      L     #WT_Nr;  //Warenträger-DB öffnen
      L     100;
      +I;
      T     #WT_DB;
      OPN   DB [#WT_DB];
      L     #WT_Nr_lang;
      T     "DB_BE_Stand".Stand[#Stand_Nr].last_WT;
      L     0;
      ==D;
      JC    noEv;

      OPN   DB [#WT_DB];
      L     0;  //Warenträger freigeben
      T     %DBD6;  //WT_Nr_lang
      T     %DBD10;  //Oberfläche
      T     %DBD18;  //Merkerfeld
      T     %DBW16;  //Technologie
      T     %DBB36;  //End_Ziel_Pos
      T     %DBB37;  //End_Ziel_Reihe
      T     %DBD46;  //Pointer
      T     %DBD50;  //SaveTime


noEv: A     #Del_All;
      O     #kein_Korb;
      JC    All;
//------------------------------------------
//Restdaten zurückladen (teilweises Löschen)
//------------------------------------------
      CALL  "FC_WT_to_Pos"
      ( Pos_Nr     := #Pos_Nr,
        WT_Nr      := #WT_Nr,
        BA_Auto    := TRUE,
        send_DBEvt := FALSE,
        SimLoad    := FALSE,
        Copy_ok    := #"Return"
      );
      BE;

//------------------------------------------
//Restdaten löschen (vollständiges Löschen)
//------------------------------------------
All:  OPN   DB [#WT_DB];  //WT bereinigen
      L     0;
      T     %DBW14;  //"DB_WTx".Korb_Nr
      BE;

END_FUNCTION

FUNCTION "FC_Hilfsfuntionen" : Void   // FC169, LAD
TITLE = Hilfsfunktionen
{ S7_Optimized_Access := 'TRUE' }
// stored: AutoNumber false, SetENOAutomatically true
   VAR_TEMP
      Anf_links : Bool;
      Anf_rechts : Bool;
      Niv_CM01_ok : Bool;
      Niv_CM02_ok : Bool;
      Niv_Spuelen_ok : Bool;
      Fuellstand_ok : Bool;
      Nr : Int;
   END_VAR
   VAR CONSTANT
      Typ_KSoLS : Byte := 16#10;
      Typ_KS : Byte := 16#11;
      Typ_LS : Byte := 16#12;
      Typ_GO_Sperre : Byte := 16#13;
      Typ_GO : Byte := 16#20;
      Ausfahrt : Byte := 16#19;
   END_VAR
BEGIN

REGION Network 1 (SCL): Einfahrsperren / Detailtypen
   REGION CM01
       // CM01 komplett leer
       IF NOT "DB_POS".POS[1].belegt AND NOT NOT "DB_POS".POS[2].belegt AND NOT "DB_POS".POS[3].belegt AND NOT "DB_POS".POS[4].belegt AND NOT "DB_POS".POS[5].belegt AND NOT "DB_POS".POS[6].belegt THEN
           "DB_POS".POS[1].notFG_in := FALSE;
           "DB_POS".POS[2].notFG_in := FALSE;
           "DB_POS".POS[5].notFG_in := FALSE;
           "DB_POS".POS[6].notFG_in := FALSE;
           "DB_POS".POS[1].Detailtyp := #Typ_KSoLS;
           "DB_POS".POS[2].Detailtyp := #Typ_KSoLS;
           "DB_POS".POS[5].Detailtyp := #Typ_KSoLS;
           "DB_POS".POS[6].Detailtyp := #Typ_KSoLS;
       END_IF;
       // Pos.3 (GO) Ziel bzw. belegt
       IF "DB_POS".POS[3].next_WT <> 0 THEN
           "DB_POS".POS[1].notFG_in := TRUE;
           "DB_POS".POS[5].notFG_in := TRUE;
           "DB_POS".POS[1].Detailtyp := #Typ_GO_Sperre;
           "DB_POS".POS[5].Detailtyp := #Typ_GO_Sperre;
       ELSE
           "DB_POS".POS[1].notFG_in := FALSE;
           "DB_POS".POS[5].notFG_in := FALSE;
           "DB_POS".POS[1].Detailtyp := #Typ_KSoLS;
           "DB_POS".POS[5].Detailtyp := #Typ_KSoLS;
       END_IF;
       // Pos.4 (GO) Ziel bzw. belegt 
       IF "DB_POS".POS[4].next_WT <> 0 THEN
           "DB_POS".POS[2].notFG_in := TRUE;
           "DB_POS".POS[6].notFG_in := TRUE;
           "DB_POS".POS[2].Detailtyp := #Typ_GO_Sperre;
           "DB_POS".POS[6].Detailtyp := #Typ_GO_Sperre;
       ELSE
           "DB_POS".POS[2].notFG_in := FALSE;
           "DB_POS".POS[6].notFG_in := FALSE;
           "DB_POS".POS[2].Detailtyp := #Typ_KSoLS;
           "DB_POS".POS[6].Detailtyp := #Typ_KSoLS;
       END_IF;
       //Pos.1/2
       IF ("DB_POS".POS[1].next_WT <> 0) AND ("DB_POS".POS[1].next_WT = "DB_POS".POS[2].next_WT) THEN
           "DB_POS".POS[1].Detailtyp := #Typ_LS;
           "DB_POS".POS[2].Detailtyp := #Typ_LS;
       ELSIF ("DB_POS".POS[1].next_WT <> 0) OR ("DB_POS".POS[2].next_WT <> 0) THEN
           "DB_POS".POS[1].Detailtyp := #Typ_KS;
           "DB_POS".POS[2].Detailtyp := #Typ_KS;
       END_IF;
       //Pos.5/6
       IF ("DB_POS".POS[5].next_WT <> 0) AND ("DB_POS".POS[5].next_WT = "DB_POS".POS[6].next_WT) THEN
           "DB_POS".POS[5].Detailtyp := #Typ_LS;
           "DB_POS".POS[6].Detailtyp := #Typ_LS;
       ELSIF ("DB_POS".POS[5].next_WT <> 0) OR ("DB_POS".POS[6].next_WT <> 0) THEN
           "DB_POS".POS[5].Detailtyp := #Typ_KS;
           "DB_POS".POS[6].Detailtyp := #Typ_KS;
       END_IF;
       //Einfahrsperre Pos.3/4
       "DB_POS".POS[3].notFG_in := ("DB_POS".POS[1].next_WT <> 0) OR ("DB_POS".POS[5].next_WT <> 0);
       "DB_POS".POS[4].notFG_in := ("DB_POS".POS[2].next_WT <> 0) OR ("DB_POS".POS[6].next_WT <> 0);
   END_REGION

   REGION CM03
       // CM03 komplett leer
       IF NOT "DB_POS".POS[7].belegt AND NOT NOT "DB_POS".POS[8].belegt AND NOT "DB_POS".POS[9].belegt AND NOT "DB_POS".POS[10].belegt AND NOT "DB_POS".POS[11].belegt AND NOT "DB_POS".POS[12].belegt THEN
           "DB_POS".POS[7].notFG_in := FALSE;
           "DB_POS".POS[8].notFG_in := FALSE;
           "DB_POS".POS[11].notFG_in := FALSE;
           "DB_POS".POS[12].notFG_in := FALSE;
           "DB_POS".POS[7].Detailtyp := #Typ_KSoLS;
           "DB_POS".POS[8].Detailtyp := #Typ_KSoLS;
           "DB_POS".POS[11].Detailtyp := #Typ_KSoLS;
           "DB_POS".POS[12].Detailtyp := #Typ_KSoLS;
       END_IF;
       // Pos.9 (GO) Ziel bzw. belegt
       IF "DB_POS".POS[9].next_WT <> 0 THEN
           "DB_POS".POS[7].notFG_in := TRUE;
           "DB_POS".POS[11].notFG_in := TRUE;
           "DB_POS".POS[7].Detailtyp := #Typ_GO_Sperre;
           "DB_POS".POS[11].Detailtyp := #Typ_GO_Sperre;
       ELSE
           "DB_POS".POS[7].notFG_in := FALSE;
           "DB_POS".POS[11].notFG_in := FALSE;
           "DB_POS".POS[7].Detailtyp := #Typ_KSoLS;
           "DB_POS".POS[11].Detailtyp := #Typ_KSoLS;
       END_IF;
       // Pos.10 (GO) Ziel bzw. belegt 
       IF "DB_POS".POS[10].next_WT <> 0 THEN
           "DB_POS".POS[8].notFG_in := TRUE;
           "DB_POS".POS[12].notFG_in := TRUE;
           "DB_POS".POS[8].Detailtyp := #Typ_GO_Sperre;
           "DB_POS".POS[12].Detailtyp := #Typ_GO_Sperre;
       ELSE
           "DB_POS".POS[8].notFG_in := FALSE;
           "DB_POS".POS[12].notFG_in := FALSE;
           "DB_POS".POS[8].Detailtyp := #Typ_KSoLS;
           "DB_POS".POS[12].Detailtyp := #Typ_KSoLS;
       END_IF;
       //Pos.7/8
       IF ("DB_POS".POS[7].next_WT <> 0) AND ("DB_POS".POS[7].next_WT = "DB_POS".POS[8].next_WT) THEN
           "DB_POS".POS[7].Detailtyp := #Typ_LS;
           "DB_POS".POS[8].Detailtyp := #Typ_LS;
       ELSIF ("DB_POS".POS[7].next_WT <> 0) OR ("DB_POS".POS[8].next_WT <> 0) THEN
           "DB_POS".POS[7].Detailtyp := #Typ_KS;
           "DB_POS".POS[8].Detailtyp := #Typ_KS;
       END_IF;
       //Pos.11/12
       IF ("DB_POS".POS[11].next_WT <> 0) AND ("DB_POS".POS[11].next_WT = "DB_POS".POS[12].next_WT) THEN
           "DB_POS".POS[11].Detailtyp := #Typ_LS;
           "DB_POS".POS[12].Detailtyp := #Typ_LS;
       ELSIF ("DB_POS".POS[11].next_WT <> 0) OR ("DB_POS".POS[12].next_WT <> 0) THEN
           "DB_POS".POS[11].Detailtyp := #Typ_KS;
           "DB_POS".POS[12].Detailtyp := #Typ_KS;
       END_IF;
       //Einfahrsperre Pos.9/10
       "DB_POS".POS[9].notFG_in := ("DB_POS".POS[7].next_WT <> 0) OR ("DB_POS".POS[11].next_WT <> 0);
       "DB_POS".POS[10].notFG_in := ("DB_POS".POS[8].next_WT <> 0) OR ("DB_POS".POS[12].next_WT <> 0);
   END_REGION

   REGION CM02
       // CM02 komplett leer
       IF NOT "DB_POS".POS[13].belegt AND NOT NOT "DB_POS".POS[14].belegt AND NOT "DB_POS".POS[15].belegt AND NOT "DB_POS".POS[16].belegt AND NOT "DB_POS".POS[17].belegt AND NOT "DB_POS".POS[18].belegt THEN
           "DB_POS".POS[13].notFG_in := FALSE;
           "DB_POS".POS[14].notFG_in := FALSE;
           "DB_POS".POS[17].notFG_in := FALSE;
           "DB_POS".POS[18].notFG_in := FALSE;
           "DB_POS".POS[13].Detailtyp := #Typ_KSoLS;
           "DB_POS".POS[14].Detailtyp := #Typ_KSoLS;
           "DB_POS".POS[17].Detailtyp := #Typ_KSoLS;
           "DB_POS".POS[18].Detailtyp := #Typ_KSoLS;
       END_IF;
       // Pos.15 (GO) Ziel bzw. belegt
       IF "DB_POS".POS[15].next_WT <> 0 THEN
           "DB_POS".POS[13].notFG_in := TRUE;
           "DB_POS".POS[17].notFG_in := TRUE;
           "DB_POS".POS[13].Detailtyp := #Typ_GO_Sperre;
           "DB_POS".POS[17].Detailtyp := #Typ_GO_Sperre;
       ELSE
           "DB_POS".POS[13].notFG_in := FALSE;
           "DB_POS".POS[17].notFG_in := FALSE;
           "DB_POS".POS[13].Detailtyp := #Typ_KSoLS;
           "DB_POS".POS[17].Detailtyp := #Typ_KSoLS;
       END_IF;
       // Pos.16 (GO) Ziel bzw. belegt 
       IF "DB_POS".POS[16].next_WT <> 0 THEN
           "DB_POS".POS[14].notFG_in := TRUE;
           "DB_POS".POS[18].notFG_in := TRUE;
           "DB_POS".POS[14].Detailtyp := #Typ_GO_Sperre;
           "DB_POS".POS[18].Detailtyp := #Typ_GO_Sperre;
       ELSE
           "DB_POS".POS[14].notFG_in := FALSE;
           "DB_POS".POS[18].notFG_in := FALSE;
           "DB_POS".POS[14].Detailtyp := #Typ_KSoLS;
           "DB_POS".POS[18].Detailtyp := #Typ_KSoLS;
       END_IF;
       //Pos.13/14
       IF ("DB_POS".POS[13].next_WT <> 0) AND ("DB_POS".POS[13].next_WT = "DB_POS".POS[14].next_WT) THEN
           "DB_POS".POS[13].Detailtyp := #Typ_LS;
           "DB_POS".POS[14].Detailtyp := #Typ_LS;
       ELSIF ("DB_POS".POS[13].next_WT <> 0) OR ("DB_POS".POS[14].next_WT <> 0) THEN
           "DB_POS".POS[13].Detailtyp := #Typ_KS;
           "DB_POS".POS[14].Detailtyp := #Typ_KS;
       END_IF;
       //Pos.17/18
       IF ("DB_POS".POS[17].next_WT <> 0) AND ("DB_POS".POS[17].next_WT = "DB_POS".POS[18].next_WT) THEN
           "DB_POS".POS[17].Detailtyp := #Typ_LS;
           "DB_POS".POS[18].Detailtyp := #Typ_LS;
       ELSIF ("DB_POS".POS[17].next_WT <> 0) OR ("DB_POS".POS[18].next_WT <> 0) THEN
           "DB_POS".POS[17].Detailtyp := #Typ_KS;
           "DB_POS".POS[18].Detailtyp := #Typ_KS;
       END_IF;
       //Einfahrsperre Pos.15/16
       "DB_POS".POS[15].notFG_in := ("DB_POS".POS[13].next_WT <> 0) OR ("DB_POS".POS[17].next_WT <> 0);
       "DB_POS".POS[16].notFG_in := ("DB_POS".POS[14].next_WT <> 0) OR ("DB_POS".POS[18].next_WT <> 0);
   END_REGION

   REGION CM04
       // CM04 komplett leer
       IF NOT "DB_POS".POS[19].belegt AND NOT NOT "DB_POS".POS[20].belegt AND NOT "DB_POS".POS[21].belegt AND NOT "DB_POS".POS[22].belegt AND NOT "DB_POS".POS[23].belegt AND NOT "DB_POS".POS[24].belegt THEN
           "DB_POS".POS[19].notFG_in := FALSE;
           "DB_POS".POS[20].notFG_in := FALSE;
           "DB_POS".POS[23].notFG_in := FALSE;
           "DB_POS".POS[24].notFG_in := FALSE;
           "DB_POS".POS[19].Detailtyp := #Typ_KSoLS;
           "DB_POS".POS[20].Detailtyp := #Typ_KSoLS;
           "DB_POS".POS[23].Detailtyp := #Typ_KSoLS;
           "DB_POS".POS[24].Detailtyp := #Typ_KSoLS;
       END_IF;
       // Pos.21 (GO) Ziel bzw. belegt
       IF "DB_POS".POS[21].next_WT <> 0 THEN
           "DB_POS".POS[19].notFG_in := TRUE;
           "DB_POS".POS[23].notFG_in := TRUE;
           "DB_POS".POS[19].Detailtyp := #Typ_GO_Sperre;
           "DB_POS".POS[23].Detailtyp := #Typ_GO_Sperre;
       ELSE
           "DB_POS".POS[19].notFG_in := FALSE;
           "DB_POS".POS[23].notFG_in := FALSE;
           "DB_POS".POS[19].Detailtyp := #Typ_KSoLS;
           "DB_POS".POS[23].Detailtyp := #Typ_KSoLS;
       END_IF;
       // Pos.22 (GO) Ziel bzw. belegt 
       IF "DB_POS".POS[22].next_WT <> 0 THEN
           "DB_POS".POS[20].notFG_in := TRUE;
           "DB_POS".POS[24].notFG_in := TRUE;
           "DB_POS".POS[20].Detailtyp := #Typ_GO_Sperre;
           "DB_POS".POS[24].Detailtyp := #Typ_GO_Sperre;
       ELSE
           "DB_POS".POS[20].notFG_in := FALSE;
           "DB_POS".POS[24].notFG_in := FALSE;
           "DB_POS".POS[20].Detailtyp := #Typ_KSoLS;
           "DB_POS".POS[24].Detailtyp := #Typ_KSoLS;
       END_IF;
       //Pos.19/20
       IF ("DB_POS".POS[19].next_WT <> 0) AND ("DB_POS".POS[19].next_WT = "DB_POS".POS[20].next_WT) THEN
           "DB_POS".POS[19].Detailtyp := #Typ_LS;
           "DB_POS".POS[20].Detailtyp := #Typ_LS;
       ELSIF ("DB_POS".POS[19].next_WT <> 0) OR ("DB_POS".POS[20].next_WT <> 0) THEN
           "DB_POS".POS[19].Detailtyp := #Typ_KS;
           "DB_POS".POS[20].Detailtyp := #Typ_KS;
       END_IF;
       //Pos.23/24
       IF ("DB_POS".POS[23].next_WT <> 0) AND ("DB_POS".POS[23].next_WT = "DB_POS".POS[24].next_WT) THEN
           "DB_POS".POS[23].Detailtyp := #Typ_LS;
           "DB_POS".POS[24].Detailtyp := #Typ_LS;
       ELSIF ("DB_POS".POS[23].next_WT <> 0) OR ("DB_POS".POS[24].next_WT <> 0) THEN
           "DB_POS".POS[23].Detailtyp := #Typ_KS;
           "DB_POS".POS[24].Detailtyp := #Typ_KS;
       END_IF;
       //Einfahrsperre Pos.21/22
       "DB_POS".POS[21].notFG_in := ("DB_POS".POS[19].next_WT <> 0) OR ("DB_POS".POS[23].next_WT <> 0);
       "DB_POS".POS[22].notFG_in := ("DB_POS".POS[20].next_WT <> 0) OR ("DB_POS".POS[24].next_WT <> 0);
   END_REGION

   REGION Übergabe
       // Übergabe komplett leer
       IF NOT "DB_POS".POS[25].belegt AND NOT NOT "DB_POS".POS[26].belegt AND NOT "DB_POS".POS[27].belegt AND NOT "DB_POS".POS[28].belegt AND NOT "DB_POS".POS[29].belegt AND NOT "DB_POS".POS[30].belegt THEN
           "DB_POS".POS[25].Detailtyp := #Typ_KSoLS;
           "DB_POS".POS[26].Detailtyp := #Typ_KSoLS;
           "DB_POS".POS[29].Detailtyp := #Typ_KSoLS;
           "DB_POS".POS[30].Detailtyp := #Typ_KSoLS;
       END_IF;
       // Pos.27 (GO) Ziel bzw. belegt
       IF "DB_POS".POS[27].next_WT <> 0 THEN
           "DB_POS".POS[25].Detailtyp := #Typ_GO_Sperre;
           "DB_POS".POS[29].Detailtyp := #Typ_GO_Sperre;
       ELSE
           "DB_POS".POS[25].Detailtyp := #Typ_KSoLS;
           "DB_POS".POS[29].Detailtyp := #Typ_KSoLS;
       END_IF;
       // Pos.22 (GO) Ziel bzw. belegt 
       IF "DB_POS".POS[28].next_WT <> 0 THEN
           "DB_POS".POS[26].Detailtyp := #Typ_GO_Sperre;
           "DB_POS".POS[30].Detailtyp := #Typ_GO_Sperre;
       ELSE
           "DB_POS".POS[26].Detailtyp := #Typ_KSoLS;
           "DB_POS".POS[30].Detailtyp := #Typ_KSoLS;
       END_IF;
       //Pos.25/26
       IF ("DB_POS".POS[25].next_WT <> 0) AND ("DB_POS".POS[25].next_WT = "DB_POS".POS[26].next_WT) THEN
           "DB_POS".POS[25].Detailtyp := #Typ_LS;
           "DB_POS".POS[26].Detailtyp := #Typ_LS;
       ELSIF ("DB_POS".POS[25].next_WT <> 0) OR ("DB_POS".POS[26].next_WT <> 0) THEN
           "DB_POS".POS[25].Detailtyp := #Typ_KS;
           "DB_POS".POS[26].Detailtyp := #Typ_KS;
       END_IF;
       //Pos.29/30
       IF ("DB_POS".POS[29].next_WT <> 0) AND ("DB_POS".POS[29].next_WT = "DB_POS".POS[30].next_WT) THEN
           "DB_POS".POS[29].Detailtyp := #Typ_LS;
           "DB_POS".POS[30].Detailtyp := #Typ_LS;
       ELSIF ("DB_POS".POS[29].next_WT <> 0) OR ("DB_POS".POS[30].next_WT <> 0) THEN
           "DB_POS".POS[29].Detailtyp := #Typ_KS;
           "DB_POS".POS[30].Detailtyp := #Typ_KS;
       END_IF;

   END_REGION
END_REGION

REGION Network 2 (SCL): Deckelanforderungen

   REGION CM01
       #Anf_links := FALSE;
       #Anf_rechts := FALSE;

       // Check Quelle
       IF ("DB_POS".POS[1].Quelle AND ("DB_POS".POS[1].WT_DB <> 0)) OR
          ("DB_POS".POS[3].Quelle AND ("DB_POS".POS[3].WT_DB <> 0)) OR
          ("DB_POS".POS[5].Quelle AND  ("DB_POS".POS[5].WT_DB <> 0)) THEN
           #Anf_links := TRUE;
       END_IF;

       IF ("DB_POS".POS[2].Quelle AND ("DB_POS".POS[2].WT_DB <> 0)) OR
           ("DB_POS".POS[4].Quelle AND ("DB_POS".POS[4].WT_DB <> 0)) OR
           ("DB_POS".POS[6].Quelle AND  ("DB_POS".POS[6].WT_DB <> 0)) THEN
           #Anf_rechts := TRUE;
       END_IF;

       IF "DB_POS".POS[1].Quelle AND ("DB_POS".POS[1].WT_DB <> 0) AND ("DB_POS".POS[1].WT_DB = "DB_POS".POS[2].WT_DB) THEN
           #Anf_rechts := TRUE;
       END_IF;

       IF "DB_POS".POS[5].Quelle AND ("DB_POS".POS[5].WT_DB <> 0) AND ("DB_POS".POS[5].WT_DB = "DB_POS".POS[6].WT_DB) THEN
           #Anf_rechts := TRUE;
       END_IF;

       // Check Ziel
       IF (("DB_POS".POS[1].Ziel AND ("DB_POS".POS[1].next_WT <> 0)) OR ("DB_POS".POS[3].Ziel AND ("DB_POS".POS[3].next_WT <> 0)) OR ("DB_POS".POS[5].Ziel AND  ("DB_POS".POS[5].next_WT <> 0))) AND "DI_FW_1".ZST.Oben_li THEN
           #Anf_links := TRUE;
       END_IF;

       IF (("DB_POS".POS[2].Ziel AND ("DB_POS".POS[2].next_WT <> 0)) OR ("DB_POS".POS[4].Ziel AND ("DB_POS".POS[4].next_WT <> 0)) OR ("DB_POS".POS[6].Ziel AND  ("DB_POS".POS[6].next_WT <> 0)))  AND "DI_FW_1".ZST.Oben_re THEN
           #Anf_rechts := TRUE;
       END_IF;

       IF "DB_POS".POS[1].Ziel AND ("DB_POS".POS[1].next_WT <> 0) AND ("DB_POS".POS[1].next_WT = "DB_POS".POS[2].next_WT)  AND "DI_FW_1".ZST.Oben_re THEN
           #Anf_rechts := TRUE;
       END_IF;

       IF "DB_POS".POS[5].Ziel AND ("DB_POS".POS[5].next_WT <> 0) AND ("DB_POS".POS[5].next_WT = "DB_POS".POS[6].next_WT)  AND "DI_FW_1".ZST.Oben_re THEN
           #Anf_rechts := TRUE;
       END_IF;
       //
       IF #Anf_links THEN
           "Deckel_CM01".Zst.Req_links_auf := TRUE;
       ELSIF "Deckel_CM01".Zst.TW_sicher THEN
           "Deckel_CM01".Zst.Req_links_auf := FALSE;
       END_IF;

       IF #Anf_rechts THEN
           "Deckel_CM01".Zst.Req_rechts_auf := TRUE;
       ELSIF "Deckel_CM01".Zst.TW_sicher THEN
           "Deckel_CM01".Zst.Req_rechts_auf := FALSE;
       END_IF;

   END_REGION

   REGION CM02
       #Anf_links := FALSE;
       #Anf_rechts := FALSE;

       // Check Quelle
       IF ("DB_POS".POS[13].Quelle AND ("DB_POS".POS[13].WT_DB <> 0)) OR
           ("DB_POS".POS[15].Quelle AND ("DB_POS".POS[15].WT_DB <> 0)) OR
           ("DB_POS".POS[17].Quelle AND  ("DB_POS".POS[17].WT_DB <> 0)) THEN
           #Anf_links := TRUE;
       END_IF;

       IF ("DB_POS".POS[14].Quelle AND ("DB_POS".POS[14].WT_DB <> 0)) OR
           ("DB_POS".POS[16].Quelle AND ("DB_POS".POS[16].WT_DB <> 0)) OR
           ("DB_POS".POS[18].Quelle AND ("DB_POS".POS[18].WT_DB <> 0)) THEN
           #Anf_rechts := TRUE;
       END_IF;

       IF "DB_POS".POS[13].Quelle AND ("DB_POS".POS[13].WT_DB <> 0) AND ("DB_POS".POS[13].WT_DB = "DB_POS".POS[14].WT_DB) THEN
           #Anf_rechts := TRUE;
       END_IF;

       IF "DB_POS".POS[17].Quelle AND ("DB_POS".POS[17].WT_DB <> 0) AND ("DB_POS".POS[17].WT_DB = "DB_POS".POS[18].WT_DB) THEN
           #Anf_rechts := TRUE;
       END_IF;

       // Check Ziel
       IF (("DB_POS".POS[13].Ziel AND ("DB_POS".POS[13].next_WT <> 0)) OR ("DB_POS".POS[15].Ziel AND ("DB_POS".POS[15].next_WT <> 0)) OR ("DB_POS".POS[17].Ziel AND  ("DB_POS".POS[17].next_WT <> 0))) AND "DI_FW_1".ZST.Oben_li THEN
           #Anf_links := TRUE;
       END_IF;

       IF (("DB_POS".POS[14].Ziel AND ("DB_POS".POS[14].next_WT <> 0)) OR ("DB_POS".POS[16].Ziel AND ("DB_POS".POS[16].next_WT <> 0)) OR ("DB_POS".POS[18].Ziel AND  ("DB_POS".POS[18].next_WT <> 0))) AND "DI_FW_1".ZST.Oben_re THEN
           #Anf_rechts := TRUE;
       END_IF;

       IF "DB_POS".POS[13].Ziel  AND ("DB_POS".POS[13].next_WT <> 0) AND ("DB_POS".POS[13].next_WT = "DB_POS".POS[14].next_WT) AND "DI_FW_1".ZST.Oben_re THEN
           #Anf_rechts := TRUE;
       END_IF;

       IF "DB_POS".POS[17].Ziel AND ("DB_POS".POS[17].next_WT <> 0) AND ("DB_POS".POS[17].next_WT = "DB_POS".POS[18].next_WT) AND "DI_FW_1".ZST.Oben_re THEN
           #Anf_rechts := TRUE;
       END_IF;
       //
       IF #Anf_links THEN
           "Deckel_CM02".Zst.Req_links_auf := TRUE;
       ELSIF "Deckel_CM02".Zst.TW_sicher THEN
           "Deckel_CM02".Zst.Req_links_auf := FALSE;
       END_IF;

       IF #Anf_rechts THEN
           "Deckel_CM02".Zst.Req_rechts_auf := TRUE;
       ELSIF "Deckel_CM02".Zst.TW_sicher THEN
           "Deckel_CM02".Zst.Req_rechts_auf := FALSE;
       END_IF;

   END_REGION
END_REGION

REGION Network 3 (SCL): Anforderung Rolltor
   "Tor".Zst.Req_Auf := ("DI_QF_WR02_03".Zst.Req_WR02_In
   OR "DI_QF_WR02_03".Zst.Req_WR03_In
   OR "DI_QF_WR02_03".Zst.Req_WR02_Out
   OR "DI_QF_WR02_03".Zst.Req_WR03_Out) AND "DI_QF_WR02_03".Zst.TW_sicher;
END_REGION

REGION Network 4 (SCL): Keine Einfahrt / kein neuer Befehl / Freigabe Ausfahrt

   // Freigabe Abluft, kein Notstrom, kein Gasalarm
   "DI_FW_Auftrag_DB".Frg_Ablauf := "DB_PNOZ_IN_Out".In.Abluft_ok AND "E_Frg_AbLW" AND "E_DL_min_ok" AND "E_Al_Gas_ok" AND NOT "E_Not-Strom" AND "E_Normal-Vers";

   //Füllstand der Becken ok, erst dann Einfahren 
   //Beide Spülbecken + 1 Säurebecken muss Niveau haben --> Signale Niveau_ok Verzögert + entsprechende Meldung
   #Niv_CM01_ok := NOT "DB_NSP".NSP[1].AM_AL_min AND "E_Niv_UeL_CM01.BL01";
   #Niv_CM02_ok := NOT "DB_NSP".NSP[13].AM_AL_min  AND  "E_Niv_UeL_CM02.BL08";
   #Niv_Spuelen_ok := NOT "DB_NSP".NSP[19].AM_AL_min;
   #Fuellstand_ok := (#Niv_CM01_ok OR #Niv_CM02_ok) AND #Niv_Spuelen_ok;

   // Kein eingeschränkter Betrieb Abluftwäscher VEW-Waser und Füllstand
   "DI_FW_Auftrag_DB".Frg_Einfahrt := "E_kein_NB_AblW" AND "DI_FW_Auftrag_DB".Frg_Ablauf AND #Fuellstand_ok AND "E_VEW_ok";

   // Freigabe Fertig-Korb 
   IF (("DB_WT1".akt_CMD = #Ausfahrt AND "DB_POS".POS["DB_WT1".POS].fertig) OR ("DB_WT2".akt_CMD = #Ausfahrt AND "DB_POS".POS["DB_WT2".POS].fertig) OR
       ("DB_WT3".akt_CMD = #Ausfahrt AND "DB_POS".POS["DB_WT3".POS].fertig) OR ("DB_WT4".akt_CMD = #Ausfahrt AND "DB_POS".POS["DB_WT4".POS].fertig) OR
       ("DB_WT5".akt_CMD = #Ausfahrt AND "DB_POS".POS["DB_WT5".POS].fertig) OR ("DB_WT6".akt_CMD = #Ausfahrt AND "DB_POS".POS["DB_WT6".POS].fertig) OR
       ("DB_WT7".akt_CMD = #Ausfahrt AND "DB_POS".POS["DB_WT7".POS].fertig) OR ("DB_WT8".akt_CMD = #Ausfahrt AND "DB_POS".POS["DB_WT8".POS].fertig) OR
       ("DB_WT9".akt_CMD = #Ausfahrt AND "DB_POS".POS["DB_WT9".POS].fertig) OR ("DB_WT10".akt_CMD = #Ausfahrt AND "DB_POS".POS["DB_WT10".POS].fertig) OR
       ("DB_WT11".akt_CMD = #Ausfahrt AND "DB_POS".POS["DB_WT11".POS].fertig) OR ("DB_WT12".akt_CMD = #Ausfahrt AND "DB_POS".POS["DB_WT12".POS].fertig))
       AND "E_T_Frg_BE"  AND "E_VEW_ok" AND "E_DL_min_ok" THEN
       "DI_FW_Auftrag_DB".Frg_Ausfahrt := TRUE;
   END_IF;
END_REGION

REGION Network 5 (SCL): Einfahsprerren CM01 / CM02
   // CM01
   "DB_POS".POS[1].Sperre_in := "Panel".CM01.Wartung;
   "DB_POS".POS[2].Sperre_in := "Panel".CM01.Wartung;
   "DB_POS".POS[3].Sperre_in := "Panel".CM01.Wartung;
   "DB_POS".POS[4].Sperre_in := "Panel".CM01.Wartung;
   "DB_POS".POS[5].Sperre_in := "Panel".CM01.Wartung;
   "DB_POS".POS[6].Sperre_in := "Panel".CM01.Wartung;

   // Übervoll (Sperre setzend - siehe NW1)
   IF NOT "E_Niv_UeL_CM01.BL01" THEN
       "DB_POS".POS[1].notFG_in := TRUE;
       "DB_POS".POS[2].notFG_in := TRUE;
       "DB_POS".POS[3].notFG_in := TRUE;
       "DB_POS".POS[4].notFG_in := TRUE;
       "DB_POS".POS[5].notFG_in := TRUE;
       "DB_POS".POS[6].notFG_in := TRUE;
   END_IF;

   // CM02
   "DB_POS".POS[13].Sperre_in := "Panel".CM02.Wartung;
   "DB_POS".POS[14].Sperre_in := "Panel".CM02.Wartung;
   "DB_POS".POS[15].Sperre_in := "Panel".CM02.Wartung;
   "DB_POS".POS[16].Sperre_in := "Panel".CM02.Wartung;
   "DB_POS".POS[17].Sperre_in := "Panel".CM02.Wartung;
   "DB_POS".POS[18].Sperre_in := "Panel".CM02.Wartung;

   // Übervoll (Sperre setzend - siehe NW1)
   IF NOT "E_Niv_UeL_CM02.BL08" THEN
       "DB_POS".POS[13].notFG_in := TRUE;
       "DB_POS".POS[14].notFG_in := TRUE;
       "DB_POS".POS[15].notFG_in := TRUE;
       "DB_POS".POS[16].notFG_in := TRUE;
       "DB_POS".POS[17].notFG_in := TRUE;
       "DB_POS".POS[18].notFG_in := TRUE;
   END_IF;
END_REGION

REGION Network 6 (SCL): Sperren Kombibetrieb GO CM02 / CM04
   IF NOT "DB_ANLAGE".config.NormalB THEN
       // CM02
       "DB_POS".POS[15].Sperre_in := TRUE;
       "DB_POS".POS[16].Sperre_in := TRUE;
       // CM04
       "DB_POS".POS[21].Sperre_in := TRUE;
       "DB_POS".POS[22].Sperre_in := TRUE;
   END_IF;
END_REGION

REGION Network 7 (SCL): Positionsincremente
   // Ungerade --> gerade

   "DB_POS".POS[2].IncPos := "DB_POS".POS[1].IncPos;
   "DB_POS".POS[4].IncPos := "DB_POS".POS[3].IncPos;
   "DB_POS".POS[6].IncPos := "DB_POS".POS[5].IncPos;
   "DB_POS".POS[8].IncPos := "DB_POS".POS[7].IncPos;
   "DB_POS".POS[10].IncPos := "DB_POS".POS[9].IncPos;
   "DB_POS".POS[12].IncPos := "DB_POS".POS[11].IncPos;
   "DB_POS".POS[14].IncPos := "DB_POS".POS[13].IncPos;
   "DB_POS".POS[16].IncPos := "DB_POS".POS[15].IncPos;
   "DB_POS".POS[18].IncPos := "DB_POS".POS[17].IncPos;
   "DB_POS".POS[20].IncPos := "DB_POS".POS[19].IncPos;
   "DB_POS".POS[22].IncPos := "DB_POS".POS[21].IncPos;
   "DB_POS".POS[24].IncPos := "DB_POS".POS[23].IncPos;
   "DB_POS".POS[26].IncPos := "DB_POS".POS[25].IncPos;
   "DB_POS".POS[28].IncPos := "DB_POS".POS[27].IncPos;
   "DB_POS".POS[30].IncPos := "DB_POS".POS[29].IncPos;
END_REGION

REGION Network 8 (SCL): Korbumläufe Meldungen
   FOR #Nr := "KorbAnzahl_min" TO "KorbAnzahl_max" DO
       IF "DB_Korbumlaeufe".Korb[#Nr].Durchlaeufe >= "DB_Korbumlaeufe".Korb[#Nr].max_Durchlaeufe THEN
           "DB_Korbumlaeufe".Korb[#Nr].max_erreicht := TRUE;
           "DB_Korbumlaeufe".Korb[#Nr].Warnung := FALSE;
       ELSIF ("DB_Korbumlaeufe".Korb[#Nr].Durchlaeufe >= ("DB_Korbumlaeufe".Korb[#Nr].max_Durchlaeufe - 3)) AND NOT "DB_Korbumlaeufe".Korb[#Nr].max_erreicht THEN
           "DB_Korbumlaeufe".Korb[#Nr].Warnung := TRUE;
       ELSE
           "DB_Korbumlaeufe".Korb[#Nr].max_erreicht := FALSE;
           "DB_Korbumlaeufe".Korb[#Nr].Warnung := FALSE;
       END_IF;
   END_FOR;
END_REGION

REGION Network 9 (SCL): Bits für Anzeige Materialcheck
   // Modus auswerten
   IF NOT "DB_ANLAGE".config.NormalB THEN
       // Kombi-Mode
       CASE "DB_Prog_edit".Prog_Aufgabe.Korb_Nr OF
           1..3:  // "151" Korb kurz 1..3
               "Panel".Betriebsmodus.Korb_151 := TRUE;
               "Panel".Betriebsmodus.Korb_161 := FALSE;

           4..8:   // "161" Korb kurz 4..8
               "Panel".Betriebsmodus.Korb_151 := FALSE;
               "Panel".Betriebsmodus.Korb_161 := TRUE;

           9..11:  // "151" Korb lang 1..3
               "Panel".Betriebsmodus.Korb_151 := TRUE;
               "Panel".Betriebsmodus.Korb_161 := FALSE;

           12..13:   // "161" Korb lang 4, Großoptik 
               "Panel".Betriebsmodus.Korb_151 := FALSE;
               "Panel".Betriebsmodus.Korb_161 := TRUE;
       END_CASE;

   ELSE
       // Normalbetrieb
       "Panel".Betriebsmodus.Korb_151 := FALSE;
       "Panel".Betriebsmodus.Korb_161 := FALSE;
   END_IF;
END_REGION
END_FUNCTION

FUNCTION "FC_FW_RES_QZ" : Void   // FC27, STL
TITLE = Reset Reserviertbits
{ S7_Optimized_Access := 'FALSE' }
AUTHOR : MS
// stored: AutoNumber false
   VAR_TEMP
      count : Int;
      DB_Nr : Int;
      B_PNTR : Int;
      newB_PNTR : Int;
      WT_DB : Int;
      adrRow : Int;
      WT_Nr : Int;
      WT_Nr_li : USInt;
      WT_Nr_re : USInt;
      Restzeit : Int;
      AdrPos : DWord;
      Pos : Byte;
      Pos2 : Byte;
      WT_Pos : USInt;
      Del_EndZiel : Bool;
      Ziel_belegt : Bool;
      amFW : Bool;
      AutoBef : Bool;
      no_UT_req : Bool;
      inA : Bool;
      outA : Bool;
      Sp_Bel : Bool;   // Speicher oder Beladepos
      ungerade : Bool;
      WT_Ziel_li : Int;
      WT_Ziel_re : Int;
   END_VAR
BEGIN

NETWORK
TITLE = Positionsdaten löschen
// Setz die Bits reservierte Quelle reserviertes ziel zurück
//------------------------------------
//Alles löschen
//------------------------------------
      SET;
      R     "DB_ANLAGE".IN.UT_Req;
      R     "DB_ANLAGE".OUT.WT_in_Anlage;
      L     0;
      T     "DB_ANLAGE".OUT.AnzUT_Req;

getP: L     "DB_ANLAGE".config.ANZ_Pos;
retP: T     #count;
      L     0;
      <=I;
      JC    dWT;
      L     #count;
      L     "DB_POS".LENG;
      *I;
      L     "DB_POS".Offset;
      +I;
      SLD   3;
      LAR1;
      OPN   "DB_POS";
      CLR;
      =     DBX [AR1, P#6.2];  //reserviert FW-Quelle
      =     DBX [AR1, P#6.3];  //reserviert FW-Ziel
      =     DBX [AR1, P#6.4];  //FW-kommt
      =     DBX [AR1, P#10.7];  //"DB_POS".POS[0].Checked

      L     0;  //Anlagenbad
      L     DBB [AR1, P#0.0];  //"DB_POS".POS[0].Typ
      <>I;
      A(;
      L     5;  //Speicherpos und Beladen zählt
      <=I;
      );
      =     #Sp_Bel;

      L     0;
      T     DBB [AR1, P#5.0];  //FW_Nr im Bad

      AN    DBX [AR1, P#96.0];  //"DB_POS".POS[0].belegt
      JC    setP;


      L     DBB [AR1, P#35.0];  //"DB_POS".POS[0].WT_DB
setP: T     DBB [AR1, P#36.0];  //"DB_POS".POS[0].next_WT


nexP: L     #count;
      LOOP  retP;

dWT:  L     "DB_ANLAGE".config.ANZ_WT;
reW:  T     #count;
      L     0;
      <=I;
      JC    endP;

      L     #count;
      +     100;
      T     #WT_DB;

//ungültige Position --> lösche WT_Nr_lang
      OPN   DB [#WT_DB];
      L     %DBB15;  //"DB_WT1".POS
      L     0;
      <>I;
      JC    WPok;
      T     %DBD6;  //"DB_WT1".WT_NR_lang

WPok: OPN   DB [#WT_DB];
      SET;
      R     %DBX20.6;  //"DB_WT1".noOPT_WT
      R     %DBX18.6;  //"DB_WT1".FW_Pos
      R     %DBX18.7;  //"DB_WT1".QT_Pos

      L     0;
      L     %DBD6;  //"DB_WT1".WT_NR_lang
      <>D;
      JC    WPos;
      L     %DBW2;  //"DB_WT1".OFFSET
      SLD   3;
      LAR1;
      L     0;
      T     DBD [AR1, P#0.0];  //Löschen erster Befehl
      T     DBD [AR1, P#4.0];
      T     %DBB36;  //"DB_WT1".End_Ziel_Pos
      T     %DBB37;  //"DB_WT1".End_Ziel_QT_Pos

WPos: L     0;
      L     %DBB36;  //"DB_WT1".End_Ziel_Pos
      ==I;
      R     %DBX20.5;  //"DB_WT1".noKorrBefx

      AN    "DB_ANLAGE".config.Anl_getaktet;
      JC    next;
      OPN   DB [#WT_DB];

      L     0;
      T     %DBB36;  //"DB_WT1".End_Ziel_Pos
      T     %DBB37;  //"DB_WT1".End_Ziel_QT_Pos

next: L     #count;
      LOOP  reW;

endP: NOP   0;

NETWORK
TITLE = Schleife über alle FW
// Positions- und WT-Informationen setzen

      L     0;
      T     #WT_Pos;

//------------------------------------
//WT-Nr laden und Bit amFW setzen
//------------------------------------
      OPN   DB [#DB_Nr];
      L     "DI_FW_1".ZST.WT_DB_NR_li;
      T     #WT_Nr_li;
      L     0;
      <>I;
      =     #amFW;

      L     "DI_FW_1".ZST.WT_DB_NR_re;
      T     #WT_Nr_re;
      L     0;
      <>I;
      S     #amFW;

      L     "DI_FW_1".ZST.BEFEHL.%B2;  //Befehlsart
      L     16#03;
      ==I;
      A     "DI_FW_1".ZST.Auto;
      =     #AutoBef;

      L     "DI_FW_1".ZST.Rest_Zeit;
      T     #Restzeit;

//FW hat WT aber keinen Befehl
// --> Daten aus WT holen und Quelle oder Ziel sperren
      A     #amFW;
      AN    #AutoBef;
      JC    SP_W;

//FW hat Befehl und WT bereits geholt
// --> WT aus Quelle holen und Quelle und Ziel sperren
      A     #amFW;
      A     #AutoBef;
      JC    SP_Z;

//FW hat Befehl aber WT noch nicht geholt
// --> WT aus Quelle holen und Quelle und Ziel sperren
      AN    #amFW;
      A     #AutoBef;
      JC    SP_Q;

//FW hat weder Befehl noch WT
// --> nächster FW
      JU    nexF;

//------------------------------------
//Quelle sperren
//------------------------------------
SP_Q: OPN   DB [#DB_Nr];
      L     0;
      L     "DI_FW_1".ZST.BEFEHL.%B1;  // Quelle
      ==I;
      JC    nexF;
      L     "DB_POS".LENG;
      *I;
      L     "DB_POS".Offset;
      +I;
      SLD   3;
      LAR1;

      L     "DI_FW_1".ZST.BEFEHL.%B1;  // Quelle
      L     2;
      MOD;
      A     <>0;
      =     #ungerade;

      OPN   "DB_POS";
      SET;
      S     DBX [AR1, P#6.2];  //reservierte Quelle

      L     DBB [AR1, P#35.0];  //WT_DB
      AN    #ungerade;
      JC    SP_Q_re;
      T     #WT_Nr_li;

      L     DBB [AR1, P#135.0];  //WT_DB
      <>I;
      JC    SP_Z;
      S     DBX [AR1, P#106.2];  //reservierte Quelle
SP_Q_re:T     #WT_Nr_re;
      JU    SP_Z;

//------------------------------------
//Ziel sperren
//------------------------------------
SP_Z: L     0;
      L     "DI_FW_1".ZST.BEFEHL.%B0;  // Ziel
      ==I;
      JC    nexF;
      L     2;
      MOD;
      A     <>0;
      L     "DI_FW_1".ZST.BEFEHL.%B0;  // Ziel
      JC    SP_Z_set;
      DEC   1;
SP_Z_set:T     #WT_Ziel_li;
      INC   1;
      T     #WT_Ziel_re;

SPWT: L     0;
      L     #WT_Ziel_li;
      ==I;
      JC    SPWT_re;
      L     "DB_POS".LENG;
      *I;
      L     "DB_POS".Offset;
      +I;
      SLD   3;
      LAR1;
      OPN   "DB_POS";
      SET;
      S     DBX [AR1, P#6.3];  //reserviertes Ziel

      L     0;
      L     #WT_Nr_li;
      >=I;
      JC    SPWT_re;

      OPN   "DB_POS";
      L     DBB [AR1, P#36.0];  //Next-WT
      L     0;
      <>I;
      JC    SPWT_re;

      L     #WT_Nr_li;
      T     DBB [AR1, P#36.0];  //Next-WT

      L     #WT_Nr_li;
      +     100;
      T     #WT_DB;

      OPN   DB [#WT_DB];
      SET;
      S     %DBX18.6;  //"DB_WT1".FW_Pos

SPWT_re:L     0;
      L     #WT_Ziel_re;
      ==I;
      JC    nexF;
      L     "DB_POS".LENG;
      *I;
      L     "DB_POS".Offset;
      +I;
      SLD   3;
      LAR1;
      OPN   "DB_POS";
      SET;
      S     DBX [AR1, P#6.3];  //reserviertes Ziel

      L     0;
      L     #WT_Nr_re;
      >=I;
      JC    nexF;

      OPN   "DB_POS";
      L     DBB [AR1, P#36.0];  //Next-WT
      L     0;
      <>I;
      JC    nexF;

      L     #WT_Nr_re;
      T     DBB [AR1, P#36.0];  //Next-WT

      L     #WT_Nr_re;
      +     100;
      T     #WT_DB;

      OPN   DB [#WT_DB];
      SET;
      S     %DBX18.6;  //"DB_WT1".FW_Pos

      JU    nexF;

//------------------------------------
//WT sperren
//------------------------------------
SP_W: L     0;
      T     #WT_Ziel_li;
      L     #WT_Nr_li;
      >=I;
      JC    SP_W_re;
      +     100;
      T     #WT_DB;

      OPN   DB [#WT_DB];
      L     0;
      L     %DBB21;  //"DB_WT1".Ziel_Pos_WT
      T     #WT_Ziel_li;
      <>I;
      JC    SP_W_re;
      L     %DBB15;
      T     #WT_Ziel_li;

SP_W_re:L     0;
      T     #WT_Ziel_re;
      L     #WT_Nr_re;
      >=I;
      JC    SPWT;
      +     100;
      T     #WT_DB;

      OPN   DB [#WT_DB];
      L     0;
      L     %DBB21;  //"DB_WT1".Ziel_Pos_WT
      T     #WT_Ziel_re;
      <>I;
      JC    SPWT;
      L     %DBB15;
      T     #WT_Ziel_re;
      JU    SPWT;

nexF: NOP   0;

endF: NOP   0;

NETWORK
TITLE = 
//------------------------------------
//WT kommt setzen
//------------------------------------
      L     "DB_ANLAGE".config.ANZ_WT;
retW: T     #count;
      L     0;
      <=I;
      JC    endW;

      L     #count;
      T     #WT_Nr;
      L     100;
      +I;
      T     #WT_DB;

//aktuellen Befehl auslesen
      OPN   DB [#WT_DB];
      L     0;
      L     %DBD6;  //"DB_WT1".WT_NR_lang
      ==D;
      T     %DBB62;  //"DB_WT1".akt_CMD
      JC    nexW;

      OPN   DB [#WT_DB];
      L     0;
      L     %DBB15;  //"DB_WT1".POS
      ==I;
      JC    nexW;
      L     %DBW48;  //"DB_WT1".B_PNTER
      L     %DBW4;  //"DB_WT1".LENG
      *D;
      L     %DBW2;  //"DB_WT1".OFFSET
      +D;
      SLD   3;
      LAR1;
      L     DBB [AR1, P#0.0];  //"DB_WT1".Befehl[x].Kennung
      T     %DBB62;  //"DB_WT1".akt_CMD

//------------------------------------
//DBB36 testen
//------------------------------------
Ncnt: OPN   DB [#WT_DB];
      A     %DBX18.6;  //"DB_WT1".FW_Pos
      O     %DBX18.7;  //"DB_WT1".QT_Pos
      JC    nexW;
      L     0;
      L     %DBB36;  //"DB_WT1".End_Ziel_Pos
      ==I;
      R     %DBX20.5;  //"DB_WT1".noKorrBefx
      JC    ckW;
      T     #WT_Pos;
      L     "DB_POS".LENG;
      *I;
      L     "DB_POS".Offset;
      +I;
      SLD   3;
      LAR1;
      OPN   "DB_POS";
      L     DBB [AR1, P#36.0];
      L     #WT_Nr;
      <>I;
      A(;
      L     DBB [AR1, P#36.0];
      L     0;
      <>I;
      );
      O(;
      L     DBB [AR1, P#0.0];  //PosTyp
      L     10;  //Typ QT
      <>I;
      A(;
      O     DBX [AR1, P#7.0];  //Sperre_in
      O     DBX [AR1, P#9.1];  //notFG_in
      );
      );
      JC    reSW;
      L     #WT_Nr;
      T     DBB [AR1, P#36.0];  //Next-WT

      CALL  "FC_FPosFree"
      ( WT_Nr    := #WT_Nr,
        Pos      := #WT_Pos,
        am_FW_QT := FALSE
      );
      JU    ckW;

reSW: OPN   DB [#WT_DB];
      L     0;
      T     %DBB36;

ckW:  L     0;
      L     %DBB15;  //"DB_WT1".POS
      ==I;
      JC    nexW;
      T     #WT_Pos;
      L     "DB_POS".LENG;
      *I;
      L     "DB_POS".Offset;
      +I;
      SLD   3;
      LAR1;
      OPN   "DB_POS";
      L     #count;
      L     DBB [AR1, P#35.0];
      ==I;
      AN    DBX [AR1, P#6.2];  //reserviert FW-Quelle
      AN    DBX [AR1, P#6.3];  //reserviert FW-Ziel
      AN    DBX [AR1, P#96.2];  //Vorruf
      AN    DBX [AR1, P#10.2];  //"DB_POS".POS[0].ignor_Exp
      A     DBX [AR1, P#6.0];  //Optipos
      A     DBX [AR1, P#6.1];  //berechnet
      JCN   ndel;
      OPN   DB [#WT_DB];
      L     0;
      T     %DBB36;  //"DB_WT1".End_Ziel_Pos
      T     %DBB37;  //"DB_WT1".End_Ziel_QT_Pos

ndel: OPN   "DB_POS";
      AN    DBX [AR1, P#9.3];  //FG_Posfree
      OPN   DB [#WT_DB];
      JC    nexW;

      CALL  "FC_FPosFree"
      ( WT_Nr    := #WT_Nr,
        Pos      := #WT_Pos,
        am_FW_QT := FALSE
      );

nexW: L     #count;
      LOOP  retW;

endW: NOP   0;
END_FUNCTION

FUNCTION "FC_FPosFree" : Void   // FC37, STL
TITLE = FPosFree weitergeben
{ S7_Optimized_Access := 'FALSE' }
AUTHOR : MS
// stored: AutoNumber false
   VAR_INPUT
      WT_Nr : Int;
      Pos : USInt;   // Position in der WT ist (sein sollte)
      am_FW_QT : Bool;
   END_VAR
   VAR_TEMP
      savAR1 : DWord;
      savAR2 : DWord;
      WT_DB : Word;
      ChkPos : Int;
      B_PNTR : Int;
      newB_PNTR : Int;
      Adresse : DWord;
      Ziel_1 : Int;
      Leng_1 : Int;
      Ziel_2 : Int;
      Leng_2 : Int;
      WT_Typ : Byte;
      Pos_Typ : Byte;
      Reihe : Byte;
      Typ_chk : Bool;   // 0=einfacher Check 10h 20h, 1=detailcheck 11h 12h usw.
      p_fnd : Bool;
      free : Bool;
      fPosfree : Bool;
   END_VAR
BEGIN

NETWORK
TITLE = Register retten
      A     "DB_ANLAGE".config.Anl_getaktet;
      BEC;

// --------------------------------
// Register retten
// --------------------------------
      TAR1;
      T     #savAR1;
      TAR2;
      T     #savAR2;

NETWORK
TITLE = Initialisierung
      L     #WT_Nr;
      +     100;
      T     #WT_DB;

      L     0;
      T     #Reihe;

NETWORK
TITLE = Zielposition prüfen
//-------------------------------------------
//Position prüfen
//-------------------------------------------
      L     #Pos;
      L     "DB_POS".LENG;
      *D;
      L     "DB_POS".Offset;
      +D;
      SLD   3;
      LAR1;
      OPN   "DB_POS";
//Pos mit anderem WT belegt --> Abbruch
      L     DBB [AR1, P#36.0];
      L     #WT_Nr;
      <>I;
      A(;
      L     DBB [AR1, P#36.0];
      L     0;
      <>I;
      );
      JC    raus;

//Pos gesperrt --> Abbruch
      L     DBB [AR1, P#0.0];  //PosTyp
      L     10;  //Typ QT
      <>I;
      A     DBX [AR1, P#9.1];  //notFG_in
      AN    #am_FW_QT;
      O     DBX [AR1, P#7.0];  //Sperre_in
      O     DBX [AR1, P#7.2];  //Sperre_out
      JC    raus;

      A     #am_FW_QT;
      S     DBX [AR1, P#6.3];  //reserviertes Ziel
      L     #WT_Nr;
      T     DBB [AR1, P#36.0];

      AN    DBX [AR1, P#9.3];  //"DB_POS".POS[0].fPosfree
      JC    raus;


NETWORK
TITLE = Initialisierung
//-------------------------------------------
//WT-Typ bestimmen (Trommel, Gestell usw.)
//-------------------------------------------
      A     "DB_ANLAGE".config.TypChckDetail;
      =     #Typ_chk;

      OPN   DB [#WT_DB];
      L     %DBB35;  //"DB_WT1".WT_Typ
      T     #WT_Typ;

//-------------------------------------------
//WT-DB öffnen
//-------------------------------------------
      L     #WT_Nr;
      L     100;
      +I;
      T     #WT_DB;
      OPN   DI [#WT_DB];
//-------------------------------------------
//Reihe bestimmen
//-------------------------------------------
      L     0;
      L     %DIB21;  //"DB_WT1".Ziel_Pos_WT
      <>I;
      JC    Reih;
      L     0;
      L     %DIB15;  //"DB_WT1".POS
      ==I;
      JC    nRh;
Reih: L     "DB_POS".LENG;
      *D;
      L     "DB_POS".Offset;
      +D;
      SLD   3;
      LAR1;
      OPN   "DB_POS";
      L     DBB [AR1, P#4.0];  //"DB_POS".POS[0].Reihe
      T     #Reihe;
//-------------------------------------------
//Befehlspointer laden
//-------------------------------------------
nRh:  L     %DIW48;  //"DB_WT1".B_PNTER
      T     #B_PNTR;

//-------------------------------------------
//Pointerkorrektur falls erforderlich
//z.Bsp: am FW oder bei DBB36<>0
//-------------------------------------------
      AN    #am_FW_QT;
      JC    endI;

      CALL  "FC_Pointer_Tech"
      ( Befehl       := #B_PNTR,
        Position     := #Pos,
        WT_Nr        := #WT_DB,
        p_fnd        := #p_fnd,
        new_Bef_Pntr := #newB_PNTR
      );

      AN    #p_fnd;
      JC    endI;

      L     #newB_PNTR;
      +     1;
      T     #B_PNTR;

endI: NOP   0;

NETWORK
TITLE = Zwngsziel prüfen
      L     #Pos;
      SLD   3;
      T     #Adresse;
      OPN   "DB_Zwangsziel";
      L     0;
      L     DBB [#Adresse];
      ==I;
      JC    endZ;
      T     #ChkPos;
      L     "DB_POS".LENG;
      *D;
      L     "DB_POS".Offset;
      +D;
      SLD   3;
      LAR1;
      OPN   "DB_POS";
      L     0;
      L     DBB [AR1, P#35.0];  //"DB_POS".POS[0].Reihe
      ==I;
      O(;
      L     #WT_Nr;
      ==I;
      );
      JC    endZ;
      L     0;
      L     DBB [AR1, P#36.0];  //"DB_POS".POS[0].Reihe
      <>I;
      A(;
      L     #WT_Nr;
      <>I;
      );
      JC    raus;

endZ: NOP   0;

NETWORK
TITLE = fPosfree-Schleife vor

      L     #B_PNTR;
retV: T     #newB_PNTR;
      OPN   DB [#WT_DB];
      L     %DBW0;  //"DB_WT1".ANZAHL
      >I;
      JC    raus;
      L     #newB_PNTR;
      L     %DBW4;  //"DB_WT1".LENG
      *D;
      L     %DBW2;  //"DB_WT1".OFFSET
      +D;
      SLD   3;
      LAR1;
      L     0;  //Ende Suchbereich
      L     DBB [AR1, P#0.0];  //"DB_WT1".Befehl[0].Kennung
      ==I;
      JC    raus;
//bis 220 normal
      L     DBB [AR1, P#0.0];  //Cmd
      L     220;
      <I;
      JC    chkB;
//220-229 (DC..E5) Variante
      L     DBB [AR1, P#0.0];  //Cmd
      L     230;
      <I;
      JC    VarB;
//230-235 (E6..EB) Quertransport
      L     DBB [AR1, P#0.0];  //Cmd
      L     240;
      <I;
      JC    nexV;
//240-249 (F0..F9) Gruppenfahrt
//250-252 (FA..FC) Speicherfahrt
      L     DBB [AR1, P#0.0];  //Cmd
      L     254;
      <I;
      JC    raus;
//254 (FE) Kontrolle//Sonderbefehle überspringen
//255 (FF) Trockner einschalten
      JU    nexV;

//Variantenbefehl
VarB: L     DBB [AR1, P#0.0];  //Cmd
      L     220;
      -I;
      T     #Ziel_1;
      +     1;
      L     "DB_Variantenbefehl".Anzahl_Varianten;
      >I;  //ungültige Variantengruppe
      JC    raus;

      OPN   DB [#WT_DB];
      L     DBW [AR1, P#6.0];  //Parameterpointer
      SLD   3;
      T     #Adresse;
      L     0;  //Variante überspringen
      L     DBB [#Adresse];  //Variante
      ==I;
      JC    nexV;
      T     #Ziel_2;
      L     "DB_Variantenbefehl".max_Var;
      >I;  //ungültige Variante
      JC    raus;

      L     #Ziel_1;
      L     "DB_Variantenbefehl".max_Var;
      *D;
      L     "DB_Variantenbefehl".Offset;
      +D;
      L     #Ziel_2;
      +D;
      +     -1;  //Korrektur Variante
      SLD   3;
      OPN   "DB_Variantenbefehl";
      T     #Adresse;

      L     DBB [#Adresse];  //Ziel_Position
VarC: T     #Ziel_1;
      L     1;
      T     #Leng_1;
      L     0;
      T     #Ziel_2;
      T     #Leng_2;

test: CALL  "FC_fPosfreePos"
      ( WT_Nr      := #WT_Nr,
        WT_Typ     := #WT_Typ,
        TypChk     := #Typ_chk,
        free       := #free,
        fPosfree   := #fPosfree,
        Zwangsziel := #ChkPos,
        Ziel_1     := #Ziel_1,
        leng_1     := #Leng_1,
        Ziel_2     := #Ziel_2,
        leng_2     := #Leng_2,
        Reihe      := #Reihe
      );

      AN    #free;
      JC    zrk;

      AN    #fPosfree;
      JC    raus;

      L     0;
      L     #ChkPos;
      ==I;
      JC    nexV;
      JU    VarC;

//Normaler Befehl
chkB: OPN   DB [#WT_DB];
      L     DBB [AR1, P#1.0];  //Ziel_1
      T     #Ziel_1;
      L     DBB [AR1, P#2.0];  //leng_1
      T     #Leng_1;
      L     DBB [AR1, P#3.0];  //Ziel_2
      T     #Ziel_2;
      L     DBB [AR1, P#4.0];  //leng_2
      T     #Leng_2;
      JU    test;

nexV: L     #newB_PNTR;
      +     1;
      JU    retV;


NETWORK
TITLE = Spuren löschen, wenn fPosfree-Strecke nicht frei
zrk:  NOP   0;
//evtl. alle Pos mit Dbb36 == WT_Nr löschen


NETWORK
TITLE = Adressregister wiederherstellen
//--------------------------------------
//Adressregister wiederherstellen
//--------------------------------------
raus: L     #savAR1;
      LAR1;
      L     #savAR2;
      LAR2;
END_FUNCTION

FUNCTION "FC_fPosfreePos" : Void   // FC128, STL
{ S7_Optimized_Access := 'FALSE' }
// stored: AutoNumber false
   VAR_INPUT
      WT_Nr : Int;
      WT_Typ : Byte;
      TypChk : Bool;
   END_VAR
   VAR_OUTPUT
      free : Bool;
      fPosfree : Bool;
      Zwangsziel : Int;
   END_VAR
   VAR_IN_OUT
      Ziel_1 : Int;
      leng_1 : Int;
      Ziel_2 : Int;
      leng_2 : Int;
      Reihe : Byte;
   END_VAR
   VAR_TEMP
      savAR1 : DWord;
      savAR2 : DWord;
      WT_DB : Word;
      ChkPos : Int;
      Adresse : DWord;
      BadTyp : Byte;
      PosTyp : Byte;
      TmpReihe : Byte;
      ZwZiel : Int;
      Leerzeit : Int;
      TmpZiel : Int;
      MemChk : Bool;
      Restzeit : DInt;
      nx_fposfree : Bool;
      temp_Free : Bool;
   END_VAR
BEGIN

NETWORK
TITLE = Register retten
// --------------------------------
// Register retten
// --------------------------------
      TAR1;
      T     #savAR1;
      TAR2;
      T     #savAR2;

NETWORK
TITLE = Initialisierung
      SET;
      S     #temp_Free;
      R     #fPosfree;
      R     #nx_fposfree;

      L     0;
      T     #Zwangsziel;
      T     #ZwZiel;
      T     #Leerzeit;
      T     #TmpZiel;

////// !!!!!!!!!!!!!!!!!!!!!!!!!!  !!!!!!!!!!!!
////// !!!!!!!!!!!!!!!!!!!!!!!!!!  !!!!!!!!!!!!
//Schleife evtl verbessern indem in Gruppen
//nach längster Leerzeit gesucht wird
////// !!!!!!!!!!!!!!!!!!!!!!!!!!  !!!!!!!!!!!!
////// !!!!!!!!!!!!!!!!!!!!!!!!!!  !!!!!!!!!!!!


NETWORK
TITLE = 
      L     #Ziel_1;
      L     "DB_POS".LENG;
      *I;
      L     "DB_POS".Offset;
      +I;
      SLD   3;
      LAR1;
      OPN   "DB_POS";
      L     DBB [AR1, P#0.0];  //"DB_POS".POS[0].Typ
      T     #BadTyp;
      L     5;  //Speichertest
      ==I;
      =     #MemChk;

retG: L     0;
      L     #leng_1;
      >=I;
      JC    nexG;
      +     -1;
      T     #leng_1;

      L     #Ziel_1;
      L     #leng_1;
      +I;
      T     #ChkPos;

      L     #ChkPos;
      L     "DB_POS".LENG;
      *D;
      L     "DB_POS".Offset;
      +D;
      SLD   3;
      LAR1;
      OPN   "DB_POS";
      L     DBB [AR1, P#0.0];  //"DB_POS".POS[0].Typ
      L     #BadTyp;  //nicht gleichen Typgruppe
      <>I;
      JC    retG;

      L     #WT_Nr;  //selbst gefunden
      L     DBB [AR1, P#36.0];  //next_WT
      ==I;
      O(;
      L     DBB [AR1, P#36.0];  //next_WT
      L     0;
      ==I;
      );
      AN    DBX [AR1, P#7.0];  //Sperre_in
      AN    DBX [AR1, P#9.1];  //notFGin
      A     DBX [AR1, P#9.3];  //FG_Posfree
      =     #nx_fposfree;

      L     0;  //Pos ist leer --> prüfen
      L     DBB [AR1, P#36.0];  //next_WT
      ==I;
      O     DBX [AR1, P#10.4];  //"DB_POS".POS[0].ignor_fPosFree
      AN    DBX [AR1, P#7.0];  //Sperre_in
      AN    DBX [AR1, P#9.1];  //notFGin
      JC    fnd;

      L     DBB [AR1, P#0.0];  //"DB_POS".POS[0].Typ
      L     0;
      ==I;
      A     DBX [AR1, P#9.1];  //notFGin
      O     DBX [AR1, P#7.0];  //Sperre_in
      JC    retG;

      L     #WT_Nr;  //selbst gefunden
      L     DBB [AR1, P#36.0];  //next_WT
      ==I;
      JC    fnd;
      JU    retG;

fnd:  OPN   "DB_POS";
      L     DBB [AR1, P#11.0];  //"DB_POS".POS[0].TrommelPos
      T     #PosTyp;

      L     #WT_Typ;  //Hi-Nibble prüfen vom WT
      AW    16#00F0;
      JZ    hiok;

      L     #PosTyp;
      AW    16#00F0;
      JZ    hiok;
      <>I;
      JC    retG;

hiok: AN    #TypChk;
      JC    WTYP;

      L     #WT_Typ;  //Lo-Nibble prüfen vom WT
      AW    16#000F;
      JZ    WTYP;

      L     #PosTyp;
      AW    16#000F;
      JZ    WTYP;
      <>I;
      JC    retG;

//-------------------------------------------
//Position reservieren
//-------------------------------------------
WTYP: A     #MemChk;
      JC    frst;
      AN    #temp_Free;
      S     #temp_Free;
      JC    frst;

      L     0;
      L     #Reihe;
      ==I;
      JC    LZC;

//------------------------------------------------
//neue Pos gleiche Reihe gemerkte Pos andere Reihe
// --> übernehmen neue Pos
//------------------------------------------------
      L     #Reihe;
      L     DBB [AR1, P#4.0];  //"DB_POS".POS[0].Reihe
      ==I;
      A(;
      L     #TmpReihe;
      L     #Reihe;
      <>I;
      );
      JC    frst;
//------------------------------------------------
//neue Pos andere Reihe gemerkte Pos gleiche Reihe
// --> übernehmen neue Pos
//------------------------------------------------
      L     #Reihe;
      L     DBB [AR1, P#4.0];  //"DB_POS".POS[0].Reihe
      <>I;
      A(;
      L     #TmpReihe;
      L     #Reihe;
      ==I;
      );
      JC    retG;
//------------------------------------------------
//bei gleichen Reihen Leerzeit berücksichtigen
//------------------------------------------------
LZC:  L     DBW [AR1, P#98.0];  //"DB_POS".POS[0].Leerzeit
      L     #Leerzeit;
      <=D;
      JC    retG;

frst: L     DBW [AR1, P#98.0];  //"DB_POS".POS[0].Leerzeit
      T     #Leerzeit;
      L     DBB [AR1, P#4.0];  //"DB_POS".POS[0].Reihe
      T     #TmpReihe;

      L     #ChkPos;
      T     #TmpZiel;
      SLD   3;
      T     #Adresse;
      OPN   "DB_Zwangsziel";
      L     0;
      L     DBB [#Adresse];
      ==I;
      T     #ZwZiel;

      A     #MemChk;
      JC    Take;

nexG: L     #Ziel_2;
      L     0;
      <>I;
      JC    wtr;
      A     #temp_Free;
      JC    Take;

      A     #nx_fposfree;
      =     #fPosfree;
      JU    raus;

wtr:  L     #Ziel_2;
      T     #Ziel_1;
      L     #leng_2;
      T     #leng_1;
      L     0;
      T     #Ziel_2;
      T     #leng_2;
      JU    retG;

Take: L     #ChkPos;
      L     "DB_POS".LENG;
      *D;
      L     "DB_POS".Offset;
      +D;
      SLD   3;
      LAR1;
      OPN   "DB_POS";
//Pos mit anderem WT belegt --> Abbruch
      L     DBB [AR1, P#36.0];
      L     #WT_Nr;
      <>I;
      A(;
      L     DBB [AR1, P#36.0];
      L     0;
      <>I;
      );
      R     #fPosfree;
      JC    raus;

//Pos gesperrt --> Abbruch
      L     DBB [AR1, P#0.0];  //PosTyp
      L     10;  //Typ QT
      <>I;
      A     DBX [AR1, P#9.1];  //notFG_in
      O     DBX [AR1, P#7.0];  //Sperre_in
      R     #fPosfree;
      JC    raus;

      L     0;
      L     DBB [AR1, P#36.0];
      <>I;
      JC    bel;
      L     #WT_Nr;
      T     DBB [AR1, P#36.0];

bel:  A     DBX [AR1, P#9.3];  //FG_Posfree
      AN    DBX [AR1, P#10.4];  //"DB_POS".POS[0].ignor_fPosFree
      AN    DBX [AR1, P#7.2];  //Sperre_out
      =     #fPosfree;

      L     #ZwZiel;
      T     #Zwangsziel;
      L     #TmpReihe;
      T     #Reihe;


NETWORK
TITLE = Adressregister wiederherstellen
//--------------------------------------
//Adressregister wiederherstellen
//--------------------------------------
raus: L     #savAR1;
      LAR1;
      L     #savAR2;
      LAR2;

NETWORK
TITLE = Ausgänge umkopieren
      A     #temp_Free;
      =     #free;

END_FUNCTION

FUNCTION_BLOCK "FB_FW_Auftrag"   // FB9, LAD
{ S7_Optimized_Access := 'TRUE' }
// stored: AutoNumber false, MemoryReserve 100, SetENOAutomatically false
   VAR
      StepNbr : Int;
      Quelle : Int;
      Ziel : Int;
      Positionen { S7_SetPoint := 'True'} : Array[1..30] of "UDT_Auftrag_Pos";
      Frg_Einfahrt { S7_SetPoint := 'True'} : Bool;
      Frg_Ausfahrt : Bool;
      Frg_Ablauf : Bool;
   END_VAR
   VAR_TEMP
      pos : Int;
      setPoint : DInt;
      WT_DB : DB_ANY;
      nextStep : Bool;
      startStep : Bool;
      parkStep : Bool;
      befehlOk : Bool;
   END_VAR
   VAR CONSTANT
      Fahrzeit : DInt := 40;
   END_VAR
BEGIN

REGION Network 1 (SCL)
   IF NOT "DI_FW_1".ZST.BEREIT OR "DI_FW_1".ZST.FEHLER OR NOT "DI_FW_1".ZST.Auto OR NOT "DI_FW_1".ZST.Unten_li OR NOT "DI_FW_1".ZST.Unten_re THEN
       RETURN;
   END_IF;
END_REGION

REGION Network 2 (SCL): Initialisierung der Werte
   FOR #pos := 1 TO 30 DO
       #Positionen[#pos].Abholbar := "DB_POS".POS[#pos].belegt AND ("DB_POS".POS[#pos].Vorruf OR "DB_POS".POS[#pos].fertig) AND NOT "DB_POS".POS[#pos].Sperre_out AND NOT "DB_POS".POS[#pos].notFG_out;
       #Positionen[#pos].Fertig := #Positionen[#pos].Abholbar AND ("DB_POS".POS[#pos].Restzeit <= #Fahrzeit);
       #Positionen[#pos].Sperre := "DB_POS".POS[#pos].belegt OR "DB_POS".POS[#pos].Sperre_in OR "DB_POS".POS[#pos].notFG_in;

       #Positionen[#pos].CheckSperre := TRUE;

       IF #Positionen[#pos].Abholbar THEN
           #setPoint := "DB_POS".POS[#pos].Soll_Expozeit;
           IF #setPoint = 0 THEN
               #setPoint := 1;
           END_IF;

           #Positionen[#pos].Oldest := DINT_TO_REAL("DB_POS".POS[#pos].Verweilzeit) / DINT_TO_REAL(#setPoint);
       ELSE
           #Positionen[#pos].Oldest := 0;
       END_IF;

       IF "DB_POS".POS[#pos].next_WT > 0 THEN
           #WT_DB := UINT_TO_DB_ANY("DB_POS".POS[#pos].next_WT + 100);
           #Positionen[#pos].Wt_Typ := #WT_DB.;
           #Positionen[#pos].Wt_Cmd := #WT_DB.;
           #Positionen[#pos].WT_151 := #WT_DB.;
       ELSE
           #Positionen[#pos].Wt_Typ := 0;
           #Positionen[#pos].Wt_Cmd := 0;
           #Positionen[#pos].WT_151 := FALSE;
       END_IF;
   END_FOR;
END_REGION

REGION Network 3 (SCL)
   CASE #StepNbr OF
       1:  // Schritt 1 CM01/CMD02 -> CM03
           IF "DB_ANLAGE".config.NormalB THEN
               "FC_FW_Auftrag_Step1_NB"(Frg_Schritt := #Frg_Ablauf,
                                        nextStep => #nextStep,
                                        startStep => #startStep,
                                        parkStep => #parkStep,
                                        Quelle := #Quelle,
                                        Ziel := #Ziel,
                                        Positionen := #Positionen);
           ELSE
               "FC_FW_Auftrag_Step1_KB"(Frg_Schritt := #Frg_Ablauf,
                                        nextStep => #nextStep,
                                        startStep => #startStep,
                                        parkStep => #parkStep,
                                        Quelle := #Quelle,
                                        Ziel := #Ziel,
                                        Positionen := #Positionen);
           END_IF;

       2:        // Schritt 1 CM03 -> CM01/CM02
           IF "DB_ANLAGE".config.NormalB THEN
               "FC_FW_Auftrag_Step2_NB"(Frg_Schritt := #Frg_Ablauf,
                                        nextStep => #nextStep,
                                        startStep => #startStep,
                                        parkStep => #parkStep,
                                        Quelle := #Quelle,
                                        Ziel := #Ziel,
                                        Positionen := #Positionen);
           ELSE
               "FC_FW_Auftrag_Step2_KB"(Frg_Schritt := #Frg_Ablauf,
                                        nextStep => #nextStep,
                                        startStep => #startStep,
                                        parkStep => #parkStep,
                                        Quelle := #Quelle,
                                        Ziel := #Ziel,
                                        Positionen := #Positionen);
           END_IF;

       3:  // Schritt 3 CM03 -> CM04
           IF "DB_ANLAGE".config.NormalB THEN
               "FC_FW_Auftrag_Step3_NB"(Frg_Schritt := #Frg_Ablauf,
                                        nextStep => #nextStep,
                                        startStep => #startStep,
                                        parkStep => #parkStep,
                                        Quelle := #Quelle,
                                        Ziel := #Ziel,
                                        Positionen := #Positionen);
           ELSE
               "FC_FW_Auftrag_Step3_KB"(Frg_Schritt := #Frg_Ablauf,
                                        nextStep => #nextStep,
                                        startStep => #startStep,
                                        parkStep => #parkStep,
                                        Quelle := #Quelle,
                                        Ziel := #Ziel,
                                        Positionen := #Positionen);
           END_IF;

       4:  // Schritt 4 WR02 -> CM03
           IF "DB_ANLAGE".config.NormalB THEN
               "FC_FW_Auftrag_Step4_NB"(Frg_Einfahrt := #Frg_Einfahrt,
                                        Frg_Schritt := #Frg_Ablauf,
                                        nextStep => #nextStep,
                                        startStep => #startStep,
                                        parkStep => #parkStep,
                                        Quelle := #Quelle,
                                        Ziel := #Ziel,
                                        Positionen := #Positionen);
           ELSE
               "FC_FW_Auftrag_Step4_KB"(Frg_Einfahrt := #Frg_Einfahrt,
                                        Frg_Schritt := #Frg_Ablauf,
                                        nextStep => #nextStep,
                                        startStep => #startStep,
                                        parkStep => #parkStep,
                                        Quelle := #Quelle,
                                        Ziel := #Ziel,
                                        Positionen := #Positionen);
           END_IF;

       5:  // Schritt 5 CM04 -> WR02
           IF  "DB_ANLAGE".config.NormalB THEN
               "FC_FW_Auftrag_Step5_NB"(Frg_Schritt := #Frg_Ablauf,
                                        nextStep => #nextStep,
                                        startStep => #startStep,
                                        parkStep => #parkStep,
                                        Quelle := #Quelle,
                                        Ziel := #Ziel,
                                        Positionen := #Positionen,
                                        Frg_Ausfahrt := #Frg_Ausfahrt);
           ELSE
               "FC_FW_Auftrag_Step5_KB"(Frg_Schritt := #Frg_Ablauf,
                                        nextStep => #nextStep,
                                        startStep => #startStep,
                                        parkStep => #parkStep,
                                        Quelle := #Quelle,
                                        Ziel := #Ziel,
                                        Positionen := #Positionen,
                                        Frg_Ausfahrt := #Frg_Ausfahrt);
           END_IF;

       6:  //Parken
           "FC_FW_Auftrag_Parken"(nextStep => #nextStep,
                                  startStep=>#startStep,
                                  Quelle := #Quelle,
                                  Ziel := #Ziel,
                                  Positionen := #Positionen);

       ELSE  // Initialisieren
           #nextStep := FALSE;
           #startStep := TRUE;
           #parkStep := FALSE;
   END_CASE;

   IF #startStep THEN
       //von vorn beginnen
       #StepNbr := 1;
   ELSIF #nextStep THEN
       //weiterschalten
       #StepNbr := #StepNbr + 1;
   ELSIF #parkStep THEN
       //parken
       #StepNbr := 6;
   ELSE
       //warten
       ;
   END_IF;
END_REGION
END_FUNCTION_BLOCK

FUNCTION_BLOCK "FB_FW_MANAGER"   // FB1, STL
{ S7_Optimized_Access := 'FALSE' }
AUTHOR : MS
// stored: AutoNumber false
   VAR_INPUT
      CallDBNr : DB_ANY;
   END_VAR
   VAR
      leng : Int := 18;
      Offset : Int := 50;
      resDW_1 : DWord;
      resDW_2 : DWord;
      resDW_3 : DWord;
      resDW_4 : DWord;
      Kettenpos : Array[1..4] of Byte;   // Positionen für Ketten (z.Bsp. Optimierungsergebnisse)
      Auto : Struct
         Anlage : Bool;
         Reihe_1 : Bool;
         Reihe_2 : Bool;
         Reihe_3 : Bool;
         Reihe_4 : Bool;
         Reihe_5 : Bool;
         res : Bool;
         res_1 : Bool;
         Anlage_not : Bool;
         Reihe_not_1 : Bool;
         Reihe_not_2 : Bool;
         Reihe_not_3 : Bool;
         Reihe_not_4 : Bool;
         Reihe_not_5 : Bool;
         res_2 : Bool;
         res_3 : Bool;
      END_STRUCT;
      resDW_6 : DWord;
      resDW_7 : DWord;
      resDW_8 : DWord;
      resDW_9 : DWord;
      resW : Int;
      akt_CT : Int;   // aktuelle SPS-Zykluszeit
      max_CT : Int;   // maximale SPS-Zykluszeit
      FW_DAT : Array[1..20] of Struct
         WT_NR_LANG : DInt;
         IST_POS : Byte;
         ZIEL_POS : Byte;
         Fahrt_Vor : Bool;
         Fahrt_Rck : Bool;
         Heben : Bool;
         Senken : Bool;
         Bereit : Bool;
         Fehler : Bool;
         Dummy : Bool;
         res : Bool;
         Tipp : Bool;
         Hand : Bool;
         Auto_Stop : Bool;
         Auto : Bool;
         Halt : Bool;
         K_Auto : Bool;
         Kette_wait_Start : Bool;
         Kette_wait_Ende : Bool;
         Unten : Bool;
         Z_Sensor : Bool;
         Oben : Bool;
         mittig : Bool;
         HWmittig : Bool;
         res_7 : Bool;
         res_8 : Bool;
         res_9 : Bool;
         WT_DB_Nr : Byte;
         IstInc : DInt;
         Stangen_Nr : Byte;
         WT_Typ : Byte;
         priorisirt : Bool;
         in_Anlage : Bool;
         in_Entmetall : Bool;
         aus_Anlage : Bool;
         aus_Entmetall : Bool;
         Speicherprog : Bool;
         Trommel : Bool;
         Leer_WT : Bool;
         BefX : Byte;
      END_STRUCT;
   END_VAR
   VAR_TEMP
      DB_Nr : Int;
      Kette_DB : Word;
      Count : Byte;
      TaktKette : Bool;
      Systime : Time;
   END_VAR
BEGIN

NETWORK
TITLE = 
//----------------------------------
//Initialisieren
//----------------------------------
      SET;
      R     #Auto.Anlage;
      R     #Auto.Reihe_1;
      R     #Auto.Anlage_not;
      R     #Auto.Reihe_not_1;

//----------------------------------
//Kommunikation zwischen FWs
      CALL  "FC_FW_Bereich";

//----------------------------------
//Rücksetzen der FW-Signale im Bad
      CALL  "FC_Reset_FWBits_im_Bad"
      ( Reset_in_out_nen := FALSE
      );


NETWORK
TITLE = Betriebsarten überprüfen
//----------------------------------
//Betriebsart-Check FW
//----------------------------------
      A     "DI_FW_1".ZST.Auto;
      S     #Auto.Anlage;
      S     #Auto.Reihe_1;
      NOT;
      S     #Auto.Anlage_not;
      S     #Auto.Reihe_not_1;


NETWORK
TITLE = FW-Bearbeitung
//----------------------------------
//FW Bearbeitung
//----------------------------------
      CALL  TIME_TCK
      ( RET_VAL := #Systime
      );

      L     #Systime;
      L     16#7FFF_FFFF;
      AD;
      T     #Systime;

      CALL  "FB_FW_x", "DI_FW_1";

//---------------------------
//FW-Bearbeitung Fahren
//---------------------------

      CALL  "FB_POS_FW_INC", "DI_FW_POS_1"
      ( SysTime := #Systime
      );

//---------------------------
//FW-Bearbeitung Heben
//---------------------------

      CALL  "FB_HUB_FW_li", "DI_FW_HUB_links"
      ( FW_DBNr := 11,
        SysTime := #Systime
      );

      CALL  "FB_HUB_FW_re", "DI_FW_HUB_rechts"
      ( FW_DBNr := 11,
        SysTime := #Systime
      );

      SET;
      R     "DI_FW_1".IN.Com_Reset;


      CALL  "FC_Reset_FWBits_im_Bad"
      ( Reset_in_out_nen := TRUE
      );

NETWORK
TITLE = FW-Schieben
//---------------------------
//Fahrwagen schieben
//---------------------------
      CALL  "FC_FW_SCHIEBEN";


NETWORK
TITLE = Querförderer
//---------------------------
//WR02 / WR03
//---------------------------
      CALL  "FB_QF", "DI_QF_WR02_03";


END_FUNCTION_BLOCK

FUNCTION "FC_FW_Bereich" : Void   // FC17, STL
TITLE = FC Datenaustausch Position FW
{ S7_Optimized_Access := 'FALSE' }
AUTHOR : MS
// Daten für gesperrten Bereich werden unter den FWs ausgetauscht.
// stored: AutoNumber false
   VAR_TEMP
      count_FW : Byte;   // Fahrwagenzählvariable
      FW_DB_vor : Word;   // FW-DB nächst höherer FW
      FW_DB_rck : Word;   // FW_DB nächst niedrigerer FW
      Abstand : DInt;
      count_Pos : Byte;
      Grenze_min : DInt;
      Grenze_max : DInt;
      Pos_loop : Bool;
   END_VAR
BEGIN

NETWORK
TITLE = Initialisierung FW Bereich
// übergibt min und max des FW-Bereichs als Initialwerte

      SET;
      S     "DI_FW_1".IN.PosGr_min;
      S     "DI_FW_1".IN.PosGr_max;

      L     "DI_FW_1".PAR.Fahrt.FAHRBEREICH_MIN;
      L     "DB_POS".LENG;
      *D;
      L     "DB_POS".Offset;
      +D;
      SLD   3;
      LAR1;
      OPN   "DB_POS";
      L     DBD [AR1, P#22.0];  //"DB_POS".POS[0].IncPos
      L     DBD [AR1, P#64.0];  //"DB_POS".POS[0].SonderPos_Offset
      -D;
      L     "DI_FW_1".PAR.Fahrt.Bereich_Pos;
      -D;
      T     "DI_FW_1".IN.Grenze_min;

      L     "DI_FW_1".PAR.Fahrt.FAHRBEREICH_MAX;
      DEC   1;  // HCA: nur unherade zählen
      L     "DB_POS".LENG;
      *D;
      L     "DB_POS".Offset;
      +D;
      SLD   3;
      LAR1;
      OPN   "DB_POS";
      L     DBD [AR1, P#22.0];  //"DB_POS".POS[0].IncPos

      L     "DI_FW_1".PAR.Fahrt.Bereich_Pos;
      +D;
      T     "DI_FW_1".IN.Grenze_max;



NETWORK
TITLE = Positionen nach Sperren absuchen
//-----------------------------------------------------
//äußere Schleife "Position"
//-----------------------------------------------------
      L     "DB_ANLAGE".config.ANZ_Pos;
retP: T     #count_Pos;
      L     1;
      <I;
      JC    endP;
      S     #Pos_loop;

      L     #count_Pos;
      L     "DB_POS".LENG;
      *D;
      L     "DB_POS".Offset;
      +D;
      SLD   3;
      LAR1;
      OPN   "DB_POS";
//-----------------------------------------------------
//Position auf Sperre prüfen
//-----------------------------------------------------
      L     DBB [AR1, P#0.0];  //Postyp QT
      L     10;
      ==I;
      A     DBX [AR1, P#9.4];  //Sperre QT
      O     DBX [AR1, P#7.1];  //Sperre FW
      JCN   nexP;
//-----------------------------------------------------
//um die Positionsmitte gesperrten Bereich aufspannen
//-----------------------------------------------------
      OPN   "DB_POS";
      L     DBD [AR1, P#22.0];  //"DB_POS".POS[0].IncPos
      L     DBW [AR1, P#28.0];  //"DB_POS".POS[0].IncAbstand_rck
      -D;
      T     #Grenze_min;
      L     DBD [AR1, P#22.0];  //"DB_POS".POS[0].IncPos
      L     DBW [AR1, P#26.0];  //"DB_POS".POS[0].IncAbstand_vor
      +D;
      T     #Grenze_max;
      JU    FWlp;
//-----------------------------------------------------
//nächste Position prüfen
//-----------------------------------------------------
nexP: L     #count_Pos;
      DEC   1;
      JU    retP;

endP: NOP   0;

NETWORK
TITLE = Bereichssperren
      L     0;
      L     "DB_Sperrbereiche".Anzahl;
      ==I;
      BEC;
retB: L     1;
      -I;
      T     #count_Pos;
      L     0;
      <I;
      BEC;
      R     #Pos_loop;

      L     #count_Pos;
      L     10;
      *D;
      L     10;
      +D;
      SLD   3;
      LAR1;
      OPN   "DB_Sperrbereiche";

      AN    DBX [AR1, P#0.0];  //"DB_Sperrbereiche".Bereich[1].aktiv
      JC    nexB;
      L     DBD [AR1, P#2.0];  //"DB_Sperrbereiche".Bereich[1].min_Inc
      T     #Grenze_min;
      L     DBD [AR1, P#6.0];  //"DB_Sperrbereiche".Bereich[1].max_Inc
      T     #Grenze_max;
      JU    FWlp;

nexB: L     #count_Pos;
      JC    retB;
      BE;

NETWORK
TITLE = FW_loop
//-----------------------------------------------------
//innere Schleife "Fahrwagen"
//-----------------------------------------------------
FWlp: L     "DB_ANLAGE".config.ANZ_FW;
retC: T     #count_FW;
      L     10;
      +I;
      T     #FW_DB_vor;
//------------------------------------------------------
//FW befindet sich links des gesperrten Bereiches
//------------------------------------------------------
      OPN   DB [#FW_DB_vor];
      L     %DBD4;  //"DI_FW_1".ZST.PosInc
      L     #Grenze_min;
      <=D;
      JC    smax;
//------------------------------------------------------
//FW befindet sich rechts des gesperrten Bereiches
//------------------------------------------------------
      L     %DBD4;  //"DI_FW_1".ZST.PosInc
      L     #Grenze_max;
      >=D;
      JC    smin;
//------------------------------------------------------
//FW befindet sich innerhalb des gesperrten Bereiches
//------------------------------------------------------
      S     %DBX53.6;  //"DI_FW_1".IN.PosGr_min
      S     %DBX53.7;  //"DI_FW_1".IN.PosGr_max
      L     #Grenze_max;
      T     %DBD54;  //"DI_FW_1".IN.Grenze_min
      L     #Grenze_min;
      T     %DBD58;  //"DI_FW_1".IN.Grenze_max
      JU    nexC;
//------------------------------------------------------
//neuen Maximalwert prüfen
//------------------------------------------------------
smax: L     %DBD58;  //"DI_FW_1".IN.Grenze_max
      >=D;
      JC    nexC;
      S     %DBX53.7;  //"DI_FW_1".IN.PosGr_max
      CAC;
      T     %DBD58;  //"DI_FW_1".IN.Grenze_max
      JU    nexC;
//------------------------------------------------------
//neuen Minimalwert prüfen
//------------------------------------------------------
smin: L     %DBD54;  //"DI_FW_1".IN.Grenze_min
      <=D;
      JC    nexC;
      S     %DBX53.6;  //"DI_FW_1".IN.PosGr_min
      CAC;
      T     %DBD54;  //"DI_FW_1".IN.Grenze_min
      JU    nexC;
//------------------------------------------------------
//nächster FW
//------------------------------------------------------
nexC: L     #count_FW;
      L     1;
      <=I;
      A     #Pos_loop;
      JC    nexP;
      L     #count_FW;
      L     1;
      <=I;
      AN    #Pos_loop;
      JC    nexB;
      -I;
      JU    retC;

END_FUNCTION

FUNCTION "FC_Reset_FWBits_im_Bad" : Void   // FC18, STL
{ S7_Optimized_Access := 'FALSE' }
AUTHOR : MS
// Setzt die Bits "FW über Bad" und "FW kommt"zurück
// stored: AutoNumber false
   VAR_INPUT
      Reset_in_out_nen : Bool;
   END_VAR
   VAR_TEMP
      anzahl : Int;
      count : Int;
      first : Bool;
   END_VAR
BEGIN

NETWORK
TITLE = 
// Schleife über alle Badpositionen
      L     "DB_ANLAGE".config.ANZ_Pos;
ret:  T     #anzahl;
      L     "DB_POS".LENG;
      *I;
      L     "DB_POS".Offset;
      +I;
      SLD   3;
      LAR1;
      OPN   "DB_POS";
//vor Bearbeitung FWs
      AN    #Reset_in_out_nen;
      R     DBX [AR1, P#6.4];  //FW kommt
      R     DBX [AR1, P#6.5];  //FW in Pos
      R     DBX [AR1, P#6.6];  //FW hebt
      R     DBX [AR1, P#6.7];  //FW senkt
//nach Bearbeitung FWs
      AN    #Reset_in_out_nen;
      JC    noGR;
      OPN   "DB_POS";
      R     DBX [AR1, P#7.3];  //FW Badbedienung nicht möglich
      R     DBX [AR1, P#96.6];  //"DB_POS".POS[0].Expo_Off
      S     #first;

noGR: L     #anzahl;
      L     1;
      <=I;
      BEC;
      L     #anzahl;
      L     1;
      -I;
      JU    ret;

END_FUNCTION

